FUNCTION_BLOCK fbOnOffDevCtrl

VAR_INPUT
	IN:BOOL;
	IN_DevName:STRING;
	In_Enable:BOOL;
	In_Reset:BOOL;


	(*Trigger*)
	In_AutoON:BOOL;
	In_OrgON:BOOL;

	(*Mechanical Interlock*)
	In_OnXLock:BOOL;

	(*Sensors*)
	In_ONSig:BOOL;

	(*Timer*)
	In_OnTON:TIME;
	in_Timeout:TIME;

END_VAR

VAR_OUTPUT
	Q:BOOL;
	Out_OnSV:BOOL;
	E_OnErr:BOOL;
	S_OnSig:BOOL;

END_VAR

VAR_IN_OUT
	
END_VAR

VAR

	(* Trigger*)
	T_ManOn:BOOL;
	T_ManOff:BOOL;

	Loc_On:BOOL;
	On_TOut: TON;
	On_TON: TON;
	Loc_OnPls: BOOL;
	OnPls: R_TRIG;
	Out_RSErr:BOOL;
	OnPosPls: F_TRIG;

END_VAR
VAR_IN_OUT

END_VAR
VAR // added by the converter: edge detectors and wires of the graphical bodies
    _w1 : BOOL;
END_VAR

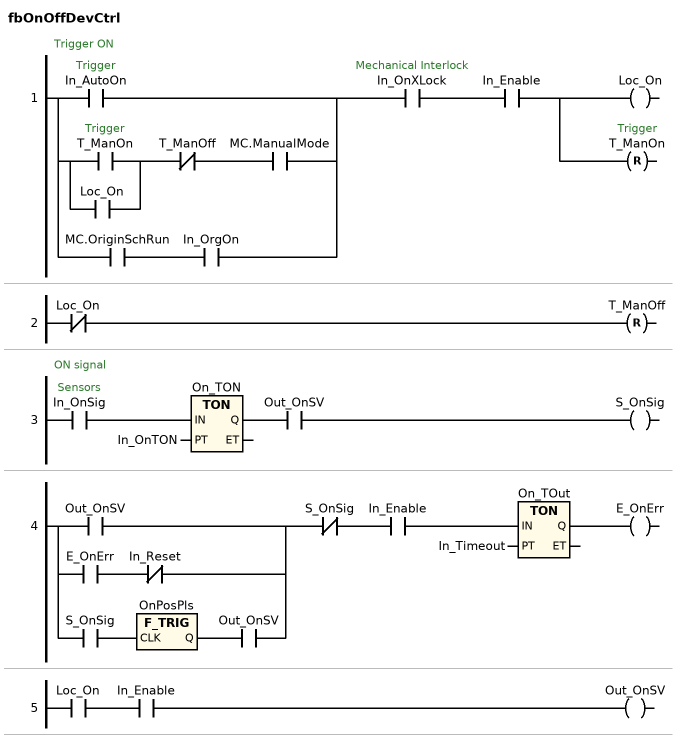
// NETWORK 1
// Trigger ON
//   In_AutoOn: Trigger
//   T_ManOn: Trigger
//   In_OnXLock: Mechanical Interlock
_w1 := (In_AutoOn OR (T_ManOn OR Loc_On) AND NOT T_ManOff AND MC.ManualMode OR MC.OriginSchRun AND In_OrgOn) AND In_OnXLock AND In_Enable;
Loc_On := _w1;
T_ManOn R= _w1;

// NETWORK 2
T_ManOff R= NOT Loc_On;

// NETWORK 3
// ON signal
//   In_OnSig: Sensors
//   In_OnTON: Timer
On_TON(IN := In_OnSig, PT := In_OnTON); // TON
S_OnSig := On_TON.Q AND Out_OnSV;

// NETWORK 4
OnPosPls(CLK := S_OnSig); // F_TRIG
On_TOut(IN := (Out_OnSV OR E_OnErr AND NOT In_Reset OR OnPosPls.Q AND Out_OnSV) AND NOT S_OnSig AND In_Enable, PT := In_Timeout); // TON
E_OnErr := On_TOut.Q;

// NETWORK 5
Out_OnSV := Loc_On AND In_Enable;

END_FUNCTION_BLOCK

(* stored: Version 1.1.0.1, ProductVersion 3.1.4018.2
   POU fbOnOffDevCtrl: Id {f24eacbe-3917-4425-a707-2cdf8e0157f7}, SpecialFunc None *)
